FUNCTION_BLOCK TestArrayList EXTENDS CNM_Collections.ArrayList
VAR_INPUT
END_VAR
VAR_OUTPUT
END_VAR
VAR
END_VAR

PROPERTY currentContainerSize : __XWORD
GET
currentContainerSize := THIS^.currentContainerCapacity;
END_GET
END_PROPERTY

END_FUNCTION_BLOCK

(* stored: Version 1.1.0.1, ProductVersion 3.1.4026.8
   POU TestArrayList: Id {7af15b8b-a788-49aa-92db-86a8ddd67e2a}, SpecialFunc None
   Property currentContainerSize: Id {486fc939-a0bd-479f-b690-55f698662aef}
   Get Get: Id {ea8a11c9-6951-4746-ae05-2ac36edec439} *)
